{attribute 'qualified_only'}
{attribute 'TcHmiSymbol' := 'true'}
VAR_GLOBAL
	
	bStartWrite : BOOL;
	bGeneratePDF: BOOL;
	bGeneratePDF2: BOOL;
	bStartRead: BOOL;
	bPreview: BOOL;
	localPDF : STRING;
	testPath : T_MaxString;
	sJsonOutput: STRING(100000);
	stReportHead: ST_ReportInfo;
	
(***** SQL Commands ***********************************************************************************)

//RUN CMDS	
isrtRun: STRING(5000) := 'INSERT INTO [dbo].[RUNS] ( [analyst], [comment], [softwareVersion], [sysMasterRevision], [sysSettingsRevision], [meterVelocity], [runVelocity], [emptyTubesFactor], [fillTubesFactor], [solvent1NameRevision], [solvent2NameRevision], [solvent3NameRevision], [solvent4NameRevision], [timeEventStarted], [timeEventCompleted], [methodID], [CalibrationNo]) VALUES ( $'#1#$', $'#2#$', $'#3#$', $'#4#$', $'#5#$', $'#6#$', $'#7#$', $'#8#$', $'#9#$', $'#10#$', $'#11#$', $'#12#$', $'#13#$', $'#14#$', $'#15#$', #16#, #17#) ';
slctLastRun: STRING(1000) := 'SELECT TOP 1 [runNo], [analyst], [comment], [softwareVersion], [sysMasterRevision], [sysSettingsRevision], [meterVelocity], [runVelocity], [emptyTubesFactor], [fillTubesFactor], [solvent1NameRevision], [solvent2NameRevision], [solvent3NameRevision], [solvent4NameRevision], [timeEventStarted], [timeEventCompleted], [methodID], [CalibrationNo] FROM [dbo].[RUNS] ORDER BY [runNo] DESC;';

//METHOD CMDS
slctAllMethods: STRING(5000) := 'SELECT [methodName], [methodRevision] FROM [dbo].[METHODS] ';
slctAllActvMethod: STRING(5000) := 'SELECT [methodName], [methodRevision] FROM [dbo].[METHODS] WHERE [methodStatus] = $'activated$'';
slctMethod: STRING(5000) := 'SELECT [methodName], [methodRevision], [methodCreatedBy], [methodCreatedOn], [solvent_R1], [solvent_R2], [solvent_W1], [solvent_W2], [time_R1], [time_R2], [time_W1], [time_W2], [velocity_R1], [velocity_R2], [velocity_W1], [velocity_W2], [soakTime], [agitate_1_Time], [agitate_2_Time], [vialsToFill], [vialPrimeVol], [vial_1_FillVol], [vial_2_4_FillVol], [airDryTime], [methodID], [methodStatus] FROM [dbo].[METHODS] WHERE [methodName] = $'#1#$' AND [methodRevision] = $'#2#$' ';
slctVD: STRING(5000) := 'SELECT [VD_ID], [pump], [stage], [rinse1], [rinse2], [wash1], [wash2], [methodID] FROM [dbo].[VOLUME_DATA] WHERE [methodID] = #1# ';
slctMethodID: STRING(5000) := 'SELECT TOP 1 [methodID] FROM [dbo].[METHODS] WHERE [methodName] = $'#1#$' ORDER BY [methodID] DESC;';
isrtNewMethod: STRING(5000) := 'INSERT INTO [dbo].[METHODS] ( [methodName], [methodRevision], [methodCreatedBy], [methodCreatedOn], [solvent_R1], [solvent_R2], [solvent_W1], [solvent_W2], [time_R1], [time_R2], [time_W1], [time_W2], [velocity_R1], [velocity_R2], [velocity_W1], [velocity_W2], [soakTime], [agitate_1_Time], [agitate_2_Time], [vialsToFill], [vialPrimeVol], [vial_1_FillVol], [vial_2_4_FillVol], [airDryTime], [methodStatus]) VALUES ( $'#1#$', $'#2#$', $'#3#$', $'#4#$', $'#5#$', $'#6#$', $'#7#$', $'#8#$', $'#9#$', $'#10#$', $'#11#$', $'#12#$', $'#13#$', $'#14#$', $'#15#$', $'#16#$', $'#17#$', $'#18#$', $'#19#$', $'#20#$', $'#21#$', $'#22#$', $'#23#$', $'#24#$', $'#25#$') ';
isrtVD: string(5000) := 'INSERT INTO [dbo].[VOLUME_DATA] ( [pump], [stage], [rinse1], [rinse2], [wash1], [wash2], [methodID]) VALUES ( $'#1#$', $'#2#$', $'#3#$', $'#4#$', $'#5#$', $'#6#$', #7#) ';
updtDactvMethod: STRING(5000) := 'UPDATE [dbo].[METHODS] SET [methodStatus] = $'deactivated$' WHERE [methodName] = $'#1#$' AND [methodRevision] = $'#2#$'';

//CALIBRATION CMD
slctLastCalibID: T_Maxstring := 'SELECT TOP 1 [calibrationNo] FROM [dbo].[CALIBRATION_HEAD] ORDER BY [calibrationNo] DESC;';
slctLastCalib: STRING(5000) := 'SELECT TOP 1 [dateTime], [pumpNo], [step], [tareWt], [grossWt], [netVolume], [netWt], [targetVolume], [differencePercent], [criteria], [pumpRevs], [CalibrationNo] FROM [dbo].[CALIBRATION] ORDER BY [calibrationNo] DESC; ';
isrtCalib: STRING(5000) := 'INSERT INTO [dbo].[CALIBRATION_HEAD] ( [userID], [density], [solventNo], [solventRevision], [allowableFail], [replicates], [callInterval], [sysRevisionNo]) VALUES ( $'#1#$', $'#2#$', $'#3#$', $'#4#$', $'#5#$', $'#6#$', $'#7#$', #8#) ';
isrtCalibValues: STRING(5000) := 'INSERT INTO [dbo].[CALIBRATION] ( [dateTime], [pumpNo], [step], [tareWt], [grossWt], [netVolume], [netWt], [targetVolume], [differencePercent], [criteria], [pumpRevs], [CalibrationNo]) VALUES ( $'#1#$', $'#2#$', $'#3#$', $'#4#$', $'#5#$', $'#6#$', $'#7#$', $'#8#$', $'#9#$', $'#10#$', $'#11#$', #12#) ';
dltCalibHead : STRING(500) :='DELETE FROM [dbo].[CALIBRATION_HEAD] WHERE [calibrationNo] = #1#';

//SYSTEM CMD
slctLastSys: STRING(5000) := 'SELECT TOP 1 [gen_SealAndPump], [cal_AcceptanceCriteria], [cal_AllowableFail], [cal_Replicates], [cal_PumpCallIntervalDays], [cal_CloseAppOnCompletation], [AirDryTimeOnCompletation], [lkt_AllowableLeakTestFail], [lkt_LeakTestBuildupTime], [lkt_LeakTestHoldTime], [lkt_LeakTestPressure], [mec_PlatesClosedPosition], [mec_PlatesDryPosition], [mec_PlatesVelocity], [mec_MaxCurrentFastDown], [mec_MaxCurrentSlowDown], [mec_MaxCurrentSlowUp], [pmp_MeterVelocity], [pmp_RunVelocity], [pmp_EmptyFactor], [pmp_FillSolventTubesFactor], [smp_AboveCalibration], [smp_VialSetSpacing], [smp_IntoResBottom], [smp_IntoResDispense], [smp_IntoResWeigh], [smp_IntoVials], [sec_DisplayManualControl], [sec_CheckLogonEachRun], [createdBy], [createdDate], [sysRevisionNo], [smp_AboveVialSet1], [smp_IntoWaste] FROM [dbo].[SYSTEM] ORDER BY [sysRevisionNo] DESC; ';
slctAllSys: STRING(5000) := 'SELECT [gen_SealAndPump], [cal_AcceptanceCriteria], [cal_AllowableFail], [cal_Replicates], [cal_PumpCallIntervalDays], [cal_CloseAppOnCompletation], [AirDryTimeOnCompletation], [lkt_AllowableLeakTestFail], [lkt_LeakTestBuildupTime], [lkt_LeakTestHoldTime], [lkt_LeakTestPressure], [mec_PlatesClosedPosition], [mec_PlatesDryPosition], [mec_PlatesVelocity], [mec_MaxCurrentFastDown], [mec_MaxCurrentSlowDown], [mec_MaxCurrentSlowUp], [pmp_MeterVelocity], [pmp_RunVelocity], [pmp_EmptyFactor], [pmp_FillSolventTubesFactor], [smp_AboveCalibration], [smp_VialSetSpacing], [smp_IntoResBottom], [smp_IntoResDispense], [smp_IntoResWeigh], [smp_IntoVials], [sec_DisplayManualControl], [sec_CheckLogonEachRun], [createdBy], [createdDate], [sysRevisionNo], [smp_AboveVialSet1], [smp_IntoWaste] FROM [dbo].[SYSTEM] ORDER BY [sysRevisionNo] DESC; ';
isrtSys: STRING(5000) := 'INSERT INTO [dbo].[SYSTEM] ( [gen_SealAndPump], [cal_AcceptanceCriteria], [cal_AllowableFail], [cal_Replicates], [cal_PumpCallIntervalDays], [cal_CloseAppOnCompletation], [AirDryTimeOnCompletation], [lkt_AllowableLeakTestFail], [lkt_LeakTestBuildupTime], [lkt_LeakTestHoldTime], [lkt_LeakTestPressure], [mec_PlatesClosedPosition], [mec_PlatesDryPosition], [mec_PlatesVelocity], [mec_MaxCurrentFastDown], [mec_MaxCurrentSlowDown], [mec_MaxCurrentSlowUp], [pmp_MeterVelocity], [pmp_RunVelocity], [pmp_EmptyFactor], [pmp_FillSolventTubesFactor], [smp_AboveCalibration], [smp_VialSetSpacing], [smp_IntoResBottom], [smp_IntoResDispense], [smp_IntoResWeigh], [smp_IntoVials], [sec_DisplayManualControl], [sec_CheckLogonEachRun], [createdBy], [createdDate], [smp_AboveVialSet1], [smp_IntoWaste]) VALUES ( $'#1#$', $'#2#$', $'#3#$', $'#4#$', $'#5#$', $'#6#$', $'#7#$', $'#8#$', $'#9#$', $'#10#$', $'#11#$', $'#12#$', $'#13#$', $'#14#$', $'#15#$', $'#16#$', $'#17#$', $'#18#$', $'#19#$', $'#20#$', $'#21#$', $'#22#$', $'#23#$', $'#24#$', $'#25#$', $'#26#$', $'#27#$', $'#28#$', $'#29#$', $'#30#$', $'#31#$', $'#32#$', $'#33#$') ';

//USERS CMD
isrtUser: STRING(5000) := 'INSERT INTO [dbo].[USERS] ( [userID], [acessLevel], [transactionType], [transactionDate], [transactedBy], [addDate], [enteredBy]) VALUES ( $'#1#$', $'#2#$', $'#3#$', $'#4#$', $'#5#$', $'#6#$', $'#7#$') ';
slctCurrentUser: STRING(5000) := 'SELECT [ID_user], [userID], [acessLevel], [transactionType], [transactionDate], [transactedBy], [addDate], [enteredBy] FROM (SELECT *, ROW_NUMBER() OVER (PARTITION BY [userID] ORDER BY TRY_CONVERT(datetime, [transactionDate], 113) DESC, [ID_user] DESC) AS rn FROM [dbo].[USERS] WHERE [transactionType] = $'Added$') t WHERE rn = 1 AND NOT EXISTS (SELECT 1 FROM [dbo].[USERS] r WHERE r.[userID] = t.[userID] AND r.[transactionType] = $'Removed$' AND TRY_CONVERT(datetime, r.[transactionDate], 113) > TRY_CONVERT(datetime, t.[transactionDate], 113));';
slctAllUsers: STRING(5000) := 'SELECT [ID_user], [userID], [acessLevel], [transactionType], [transactionDate], [transactedBy], [addDate], [enteredBy] FROM [dbo].[USERS] ';

//SOLVENTS
isrtSolvent: STRING(1000) := 'INSERT INTO [dbo].[SOLVENTS] ( [solventName1], [solventName2], [solventName3], [solventName4], [density1], [density2], [density3], [density4], [addedBy], [addedDate]) VALUES ( $'#1#$', $'#2#$', $'#3#$', $'#4#$', $'#5#$', $'#6#$', $'#7#$', $'#8#$', $'#9#$', $'#10#$') ';
slctSolvent: STRING(1000) := 'SELECT TOP 1 [SOLVENT_ID], [solventName1], [solventName2], [solventName3], [solventName4], [density1], [density2], [density3], [density4], [addedBy], [addedDate] FROM [dbo].[SOLVENTS] ORDER BY [SOLVENT_ID] DESC; ';
slctAllSolvents: STRING(1000) := 'SELECT [SOLVENT_ID], [solventName1], [solventName2], [solventName3], [solventName4], [density1], [density2], [density3], [density4], [addedBy], [addedDate] FROM [dbo].[SOLVENTS] ';

//LINEAR MOTORS
isrtLinear: STRING(1500) := 'INSERT INTO [dbo].[LINEAR] ( [pump1], [pump2], [pump3], [pump4], [pump5], [pump6], [pump7], [pump8], [pump9], [pump10], [changedBy], [changedOn]) VALUES ( $'#1#$', $'#2#$', $'#3#$', $'#4#$', $'#5#$', $'#6#$', $'#7#$', $'#8#$', $'#9#$', $'#10#$', $'#11#$', $'#12#$') ';
slctLinear: STRING(1000) := 'SELECT TOP 1 [ID_Linear], [pump1], [pump2], [pump3], [pump4], [pump5], [pump6], [pump7], [pump8], [pump9], [pump10] FROM [dbo].[LINEAR] ORDER BY [ID_Linear] DESC; ';

//PUMP CALIBRATION REPORT / HISTORY CMD
slctCalibReportList: STRING(5000) := 'SELECT TOP 50 [CalibrationNo], [userID], [solventNo], [sysRevisionNo] FROM [dbo].[PumpCalibrationHeader] ORDER BY [CalibrationNo] DESC;';
slctPumpCalibHeaderByNo: STRING(5000) := 'SELECT TOP 1 [CalibrationNo], [userID], [density], [solventNo], [solventRevision], [allowableFail], [replicates], [callInterval], [sysRevisionNo] FROM [dbo].[PumpCalibrationHeader] WHERE [CalibrationNo] = #1#;';
slctPumpCalibValuesByNo: STRING(5000) := 'SELECT [CalibrationNo], [dateTime], [pumpNo], [step], [tareWt], [grossWt], [netVolume], [netWt], [targetVolume], [differencePercent], [criteria], [pumpRevs] FROM [dbo].[PumpCalibrationValues] WHERE [CalibrationNo] = #1# ORDER BY [ID] ASC;';

slctCalibReportListFromValues: STRING(5000) := 'SELECT TOP 100 CAST(ISNULL([ReportType], $'$') AS VARCHAR(50)) AS [ReportType], CAST(ISNULL([ReportID], $'$') AS VARCHAR(50)) AS [ReportID], CAST(ISNULL([CreatedOn], $'$') AS VARCHAR(30)) AS [CreatedOn], CAST(ISNULL([CreatedBy], $'$') AS VARCHAR(50)) AS [CreatedBy], CAST(ISNULL([Description], $'$') AS VARCHAR(200)) AS [Description], CAST(ISNULL([sPrimaryKey], $'$') AS VARCHAR(50)) AS [sPrimaryKey] FROM [dbo].[vw_ReportList_PumpCalibration] ORDER BY CAST([ReportID] AS INT) DESC;';
slctMethodReportList: STRING(5000) := 'SELECT TOP 50 $'Method$' AS [ReportType], CAST([methodID] AS VARCHAR(50)) AS [ReportID], [methodCreatedOn] AS [CreatedOn], [methodCreatedBy] AS [CreatedBy], [methodName] + $' Rev $' + [methodRevision] AS [Description], CAST([methodID] AS VARCHAR(50)) AS [sPrimaryKey] FROM [dbo].[METHODS] ORDER BY [methodID] DESC;';
slctRunReportList: STRING(5000) := 'SELECT TOP 100 CAST(ISNULL($'Run$', $'$') AS VARCHAR(50)) AS [ReportType], CAST(ISNULL(CAST([runNo] AS VARCHAR(50)), $'$') AS VARCHAR(50)) AS [ReportID], CAST(ISNULL([timeEventCompleted], $'$') AS VARCHAR(30)) AS [CreatedOn], CAST(ISNULL([analyst], $'$') AS VARCHAR(50)) AS [CreatedBy], CAST(ISNULL($'Method ID $' + CAST([methodID] AS VARCHAR(20)) + $' / Cal $' + CAST([CalibrationNo] AS VARCHAR(20)) + CASE WHEN ISNULL([comment], $'$') = $'$' THEN $'$' ELSE $' - $' + [comment] END, $'$') AS VARCHAR(200)) AS [Description], CAST(ISNULL(CAST([runNo] AS VARCHAR(50)), $'$') AS VARCHAR(50)) AS [sPrimaryKey] FROM [dbo].[RUNS] ORDER BY [runNo] DESC;';
slctLinearReportList: STRING(5000) := 'SELECT TOP 50 $'Linear$' AS [ReportType], CAST([ID_Linear] AS VARCHAR(50)) AS [ReportID], $'$' AS [CreatedOn], $'$' AS [CreatedBy], $'Linear pump positions set $' + CAST([ID_Linear] AS VARCHAR(20)) AS [Description], CAST([ID_Linear] AS VARCHAR(50)) AS [sPrimaryKey] FROM [dbo].[LINEAR] ORDER BY [ID_Linear] DESC;';

// REPORT SCREEN LISTING AND SELECTING
slctPumpCalibHeaderByNo1: STRING(5000) := 'SELECT TOP 1 CAST($'Pump Calibration$' AS VARCHAR(50)) AS [sReportId], CAST(ISNULL([CalibrationNo], $'$') AS VARCHAR(30)) AS [sCalibrationNo], CAST(ISNULL([userID], $'$') AS VARCHAR(50)) AS [sUserId], CAST(ISNULL([density], $'$') AS VARCHAR(30)) AS [sDensity], CAST(ISNULL([solventNo], $'$') AS VARCHAR(30)) AS [sSolventNo], CAST(ISNULL([solventRevision], $'$') AS VARCHAR(30)) AS [sSolventRevision], CAST(ISNULL([sysRevisionNo], $'$') AS VARCHAR(30)) AS [sSysRevisionNo], CAST(ISNULL([allowableFail], $'$') AS VARCHAR(30)) AS [sAllowableFail], CAST(ISNULL([replicates], $'$') AS VARCHAR(30)) AS [sReplicates], CAST(ISNULL([callInterval], $'$') AS VARCHAR(30)) AS [sCallInterval], CAST($'$' AS VARCHAR(30)) AS [sCreatedAt] FROM [dbo].[CALIBRATION_HEAD] WHERE [CalibrationNo] = #1#;';
slctPumpCalibValuesByNo1: STRING(5000) := 'SELECT CAST(ISNULL([dateTime], $'$') AS VARCHAR(40)) AS [sDateTime], CAST(ISNULL([pumpNo], $'$') AS VARCHAR(10)) AS [sPumpNo], CAST(ISNULL([step], $'$') AS VARCHAR(20)) AS [sStep], CAST(ISNULL([tareWt], $'$') AS VARCHAR(30)) AS [sTareWt], CAST(ISNULL([grossWt], $'$') AS VARCHAR(30)) AS [sGrossWt], CAST(ISNULL([netWt], $'$') AS VARCHAR(30)) AS [sNetWt], CAST(ISNULL([netVolume], $'$') AS VARCHAR(30)) AS [sNetVolume], CAST(ISNULL([targetVolume], $'$') AS VARCHAR(30)) AS [sTargetVolume], CAST(ISNULL([differencePercent], $'$') AS VARCHAR(30)) AS [sDifferencePercent], CAST(ISNULL([criteria], $'$') AS VARCHAR(20)) AS [sCriteria], CAST(ISNULL([pumpRevs], $'$') AS VARCHAR(30)) AS [sPumpRevs] FROM [dbo].[CALIBRATION] WHERE [CalibrationNo] = #1# ORDER BY [Data_ID] ASC;';
slctSystemSettingsReportList: STRING(5000) := 'SELECT TOP 100 CAST([ReportType] AS VARCHAR(50)) AS [ReportType], CAST([ReportID] AS VARCHAR(50)) AS [ReportID], CAST([CreatedOn] AS VARCHAR(30)) AS [CreatedOn], CAST([CreatedBy] AS VARCHAR(50)) AS [CreatedBy], CAST([Description] AS VARCHAR(200)) AS [Description], CAST([sPrimaryKey] AS VARCHAR(50)) AS [sPrimaryKey] FROM [dbo].[vw_ReportList_SystemSettings] ORDER BY CAST([ReportID] AS INT) DESC;';
slctSystemSettingsByRevision: STRING(5000) := 'SELECT TOP 1 CAST([gen_SealAndPump] AS VARCHAR(100)) AS [sGenSealAndPump], CAST([cal_AcceptanceCriteria] AS VARCHAR(100)) AS [sCalAcceptanceCriteria], CAST([cal_AllowableFail] AS VARCHAR(100)) AS [sCalAllowableFail], CAST([cal_Replicates] AS VARCHAR(100)) AS [sCalReplicates], CAST([cal_PumpCallIntervalDays] AS VARCHAR(100)) AS [sCalPumpCallIntervalDays], CAST([cal_CloseAppOnCompletation] AS VARCHAR(100)) AS [sCalCloseAppOnCompletion], CAST([AirDryTimeOnCompletation] AS VARCHAR(100)) AS [sAirDryTimeOnCompletion], CAST([lkt_AllowableLeakTestFail] AS VARCHAR(100)) AS [sLktAllowableLeakTestFail], CAST([lkt_LeakTestBuildupTime] AS VARCHAR(100)) AS [sLktLeakTestBuildUpTime], CAST([lkt_LeakTestHoldTime] AS VARCHAR(100)) AS [sLktLeakTestHoldTime], CAST([lkt_LeakTestPressure] AS VARCHAR(100)) AS [sLktLeakTestPressure], CAST([mec_PlatesClosedPosition] AS VARCHAR(100)) AS [sMecPlatesClosedPosition], CAST([mec_PlatesDryPosition] AS VARCHAR(100)) AS [sMecPlatesDryPosition], CAST([mec_PlatesVelocity] AS VARCHAR(100)) AS [sMecPlatesVelocity], CAST([mec_MaxCurrentFastDown] AS VARCHAR(100)) AS [sMecMaxCurrentFastDown], CAST([mec_MaxCurrentSlowDown] AS VARCHAR(100)) AS [sMecMaxCurrentSlowDown], CAST([mec_MaxCurrentSlowUp] AS VARCHAR(100)) AS [sMecMaxCurrentSlowUp], CAST([pmp_MeterVelocity] AS VARCHAR(100)) AS [sPmpMeterVelocity], CAST([pmp_RunVelocity] AS VARCHAR(100)) AS [sPmpRunVelocity], CAST([pmp_EmptyFactor] AS VARCHAR(100)) AS [sPmpEmptyFactor], CAST([pmp_FillSolventTubesFactor] AS VARCHAR(100)) AS [sPmpFillSolventTubesFactor], CAST([smp_AboveCalibration] AS VARCHAR(100)) AS [sSmpAboveCalibration], CAST([smp_VialSetSpacing] AS VARCHAR(100)) AS [sSmpVialSetSpacing], CAST([smp_IntoResBottom] AS VARCHAR(100)) AS [sSmpIntoResBottom], CAST([smp_IntoResDispense] AS VARCHAR(100)) AS [sSmpIntoResDispense], CAST([smp_IntoResWeigh] AS VARCHAR(100)) AS [sSmpIntoResWeigh], CAST([smp_IntoVials] AS VARCHAR(100)) AS [sSmpIntoVials], CAST([smp_IntoWaste] AS VARCHAR(100)) AS [sSmpIntoWaste], CAST([sec_DisplayManualControl] AS VARCHAR(100)) AS [sSecDisplayManualControl], CAST([sec_CheckLogonEachRun] AS VARCHAR(100)) AS [sSecCheckLogonEachRun], CAST([createdBy] AS VARCHAR(100)) AS [sCreatedBy], CAST([createdDate] AS VARCHAR(100)) AS [sCreatedDate], CAST([sysRevisionNo] AS VARCHAR(30)) AS [sSysRevisionNo] FROM [dbo].[SYSTEM] WHERE [sysRevisionNo] = #1#;';
slctMethodReportSearchLatest : STRING(5000) := 'SELECT TOP 100 CAST(ISNULL([ReportType], $'$') AS VARCHAR(50)) AS [ReportType], CAST(ISNULL([ReportID], $'$') AS VARCHAR(50)) AS [ReportID], CAST(ISNULL([CreatedOn], $'$') AS VARCHAR(30)) AS [CreatedOn], CAST(ISNULL([CreatedBy], $'$') AS VARCHAR(50)) AS [CreatedBy], CAST(ISNULL([Description], $'$') AS VARCHAR(200)) AS [Description], CAST(ISNULL([sPrimaryKey], $'$') AS VARCHAR(50)) AS [sPrimaryKey] FROM [dbo].[vw_ReportList_Recipe] ORDER BY CAST([ReportID] AS INT) DESC;';
slctMethodHeaderByID : STRING(5000) := 'SELECT TOP 1 CAST(ISNULL([methodName], $'$') AS VARCHAR(100)) AS [methodName], CAST(ISNULL([methodRevision], $'$') AS VARCHAR(100)) AS [methodRevision], CAST(ISNULL([methodCreatedBy], $'$') AS VARCHAR(100)) AS [methodCreatedBy], CAST(ISNULL([methodCreatedOn], $'$') AS VARCHAR(100)) AS [methodCreatedOn], CAST(ISNULL([solvent_R1], $'$') AS VARCHAR(100)) AS [solvent_R1], CAST(ISNULL([solvent_R2], $'$') AS VARCHAR(100)) AS [solvent_R2], CAST(ISNULL([solvent_W1], $'$') AS VARCHAR(100)) AS [solvent_W1], CAST(ISNULL([solvent_W2], $'$') AS VARCHAR(100)) AS [solvent_W2], CAST(ISNULL([time_R1], $'$') AS VARCHAR(100)) AS [time_R1], CAST(ISNULL([time_R2], $'$') AS VARCHAR(100)) AS [time_R2], CAST(ISNULL([time_W1], $'$') AS VARCHAR(100)) AS [time_W1], CAST(ISNULL([time_W2], $'$') AS VARCHAR(100)) AS [time_W2], CAST(ISNULL([velocity_R1], $'$') AS VARCHAR(100)) AS [velocity_R1], CAST(ISNULL([velocity_R2], $'$') AS VARCHAR(100)) AS [velocity_R2], CAST(ISNULL([velocity_W1], $'$') AS VARCHAR(100)) AS [velocity_W1], CAST(ISNULL([velocity_W2], $'$') AS VARCHAR(100)) AS [velocity_W2], CAST(ISNULL([soakTime], $'$') AS VARCHAR(100)) AS [soakTime], CAST(ISNULL([agitate_1_Time], $'$') AS VARCHAR(100)) AS [agitate_1_Time], CAST(ISNULL([agitate_2_Time], $'$') AS VARCHAR(100)) AS [agitate_2_Time], CAST(ISNULL([vialsToFill], $'$') AS VARCHAR(100)) AS [vialsToFill], CAST(ISNULL([vialPrimeVol], $'$') AS VARCHAR(100)) AS [vialPrimeVol], CAST(ISNULL([vial_1_FillVol], $'$') AS VARCHAR(100)) AS [vial_1_FillVol], CAST(ISNULL([vial_2_4_FillVol], $'$') AS VARCHAR(100)) AS [vial_2_4_FillVol], CAST(ISNULL([airDryTime], $'$') AS VARCHAR(100)) AS [airDryTime], ISNULL([methodID], 0) AS [methodID], CAST(ISNULL([methodStatus], $'$') AS VARCHAR(100)) AS [methodStatus] FROM [dbo].[METHODS] WHERE [methodID] = #1#;';
slctMethodVolumeByID : STRING(5000) := 'SELECT ISNULL([VD_ID], 0) AS [VD_ID], CAST(ISNULL([pump], $'$') AS VARCHAR(100)) AS [pump], CAST(ISNULL([stage], $'$') AS VARCHAR(100)) AS [stage], CAST(ISNULL([rinse1], $'$') AS VARCHAR(100)) AS [rinse1], CAST(ISNULL([rinse2], $'$') AS VARCHAR(100)) AS [rinse2], CAST(ISNULL([wash1], $'$') AS VARCHAR(100)) AS [wash1], CAST(ISNULL([wash2], $'$') AS VARCHAR(100)) AS [wash2], ISNULL([methodID], 0) AS [methodID] FROM [dbo].[VOLUME_DATA] WHERE [methodID] = #1# ORDER BY [VD_ID] ASC;';
slctPostRunHeaderByID : STRING(5000) := 'SELECT TOP 1 ISNULL([runNo], 0) AS [runNo], CAST(ISNULL([analyst], $'$') AS VARCHAR(100)) AS [analyst], CAST(ISNULL([comment], $'$') AS VARCHAR(100)) AS [comment], CAST(ISNULL([softwareVersion], $'$') AS VARCHAR(100)) AS [softwareVersion], CAST(ISNULL([sysMasterRevision], $'$') AS VARCHAR(100)) AS [sysMasterRevision], CAST(ISNULL([sysSettingsRevision], $'$') AS VARCHAR(100)) AS [sysSettingsRevision], CAST(ISNULL([meterVelocity], $'$') AS VARCHAR(100)) AS [meterVelocity], CAST(ISNULL([runVelocity], $'$') AS VARCHAR(100)) AS [runVelocity], CAST(ISNULL([emptyTubesFactor], $'$') AS VARCHAR(100)) AS [emptyTubesFactor], CAST(ISNULL([fillTubesFactor], $'$') AS VARCHAR(100)) AS [fillTubesFactor], CAST(ISNULL([solvent1NameRevision], $'$') AS VARCHAR(100)) AS [solvent1NameRevision], CAST(ISNULL([solvent2NameRevision], $'$') AS VARCHAR(100)) AS [solvent2NameRevision], CAST(ISNULL([solvent3NameRevision], $'$') AS VARCHAR(100)) AS [solvent3NameRevision], CAST(ISNULL([solvent4NameRevision], $'$') AS VARCHAR(100)) AS [solvent4NameRevision], CAST(ISNULL([timeEventStarted], $'$') AS VARCHAR(100)) AS [timeEventStarted], CAST(ISNULL([timeEventCompleted], $'$') AS VARCHAR(100)) AS [timeEventCompleted], ISNULL([methodID], 0) AS [methodID], ISNULL([CalibrationNo], 0) AS [CalibrationNo] FROM [dbo].[RUNS] WHERE [runNo] = #1#;';
slctPostRunMethodHeaderByID : STRING(5000) := 'SELECT TOP 1 CAST(ISNULL([methodName], $'$') AS VARCHAR(100)) AS [methodName], CAST(ISNULL([methodRevision], $'$') AS VARCHAR(100)) AS [methodRevision], CAST(ISNULL([methodCreatedBy], $'$') AS VARCHAR(100)) AS [methodCreatedBy], CAST(ISNULL([methodCreatedOn], $'$') AS VARCHAR(100)) AS [methodCreatedOn], CAST(ISNULL([solvent_R1], $'$') AS VARCHAR(100)) AS [solvent_R1], CAST(ISNULL([solvent_R2], $'$') AS VARCHAR(100)) AS [solvent_R2], CAST(ISNULL([solvent_W1], $'$') AS VARCHAR(100)) AS [solvent_W1], CAST(ISNULL([solvent_W2], $'$') AS VARCHAR(100)) AS [solvent_W2], CAST(ISNULL([time_R1], $'$') AS VARCHAR(100)) AS [time_R1], CAST(ISNULL([time_R2], $'$') AS VARCHAR(100)) AS [time_R2], CAST(ISNULL([time_W1], $'$') AS VARCHAR(100)) AS [time_W1], CAST(ISNULL([time_W2], $'$') AS VARCHAR(100)) AS [time_W2], CAST(ISNULL([velocity_R1], $'$') AS VARCHAR(100)) AS [velocity_R1], CAST(ISNULL([velocity_R2], $'$') AS VARCHAR(100)) AS [velocity_R2], CAST(ISNULL([velocity_W1], $'$') AS VARCHAR(100)) AS [velocity_W1], CAST(ISNULL([velocity_W2], $'$') AS VARCHAR(100)) AS [velocity_W2], CAST(ISNULL([soakTime], $'$') AS VARCHAR(100)) AS [soakTime], CAST(ISNULL([agitate_1_Time], $'$') AS VARCHAR(100)) AS [agitate_1_Time], CAST(ISNULL([agitate_2_Time], $'$') AS VARCHAR(100)) AS [agitate_2_Time], CAST(ISNULL([vialsToFill], $'$') AS VARCHAR(100)) AS [vialsToFill], CAST(ISNULL([vialPrimeVol], $'$') AS VARCHAR(100)) AS [vialPrimeVol], CAST(ISNULL([vial_1_FillVol], $'$') AS VARCHAR(100)) AS [vial_1_FillVol], CAST(ISNULL([vial_2_4_FillVol], $'$') AS VARCHAR(100)) AS [vial_2_4_FillVol], CAST(ISNULL([airDryTime], $'$') AS VARCHAR(100)) AS [airDryTime], ISNULL([methodID], 0) AS [methodID], CAST(ISNULL([methodStatus], $'$') AS VARCHAR(100)) AS [methodStatus] FROM [dbo].[METHODS] WHERE [methodID] = #1#;';
slctPostRunVolumeByMethodID : STRING(5000) := 'SELECT ISNULL([VD_ID], 0) AS [VD_ID], CAST(ISNULL([pump], $'$') AS VARCHAR(100)) AS [pump], CAST(ISNULL([stage], $'$') AS VARCHAR(100)) AS [stage], CAST(ISNULL([rinse1], $'$') AS VARCHAR(100)) AS [rinse1], CAST(ISNULL([rinse2], $'$') AS VARCHAR(100)) AS [rinse2], CAST(ISNULL([wash1], $'$') AS VARCHAR(100)) AS [wash1], CAST(ISNULL([wash2], $'$') AS VARCHAR(100)) AS [wash2], ISNULL([methodID], 0) AS [methodID] FROM [dbo].[VOLUME_DATA] WHERE [methodID] = #1# ORDER BY [VD_ID] ASC;';
slctLinearReportSearch : STRING(5000) := 'SELECT TOP 100 CAST(ISNULL([ReportType], $'$') AS VARCHAR(50)) AS [ReportType], CAST(ISNULL([ReportID], $'$') AS VARCHAR(50)) AS [ReportID], CAST(ISNULL([CreatedOn], $'$') AS VARCHAR(30)) AS [CreatedOn], CAST(ISNULL([CreatedBy], $'$') AS VARCHAR(50)) AS [CreatedBy], CAST(ISNULL([Description], $'$') AS VARCHAR(200)) AS [Description], CAST(ISNULL([sPrimaryKey], $'$') AS VARCHAR(50)) AS [sPrimaryKey] FROM [dbo].[vw_ReportList_Linear] ORDER BY CAST([ReportID] AS INT) DESC;';
slctLinearByID : STRING(5000) := 'SELECT TOP 1 ISNULL([ID_Linear], 0) AS [ID_Linear], CAST(ISNULL([pump1], $'$') AS VARCHAR(100)) AS [pump1], CAST(ISNULL([pump2], $'$') AS VARCHAR(100)) AS [pump2], CAST(ISNULL([pump3], $'$') AS VARCHAR(100)) AS [pump3], CAST(ISNULL([pump4], $'$') AS VARCHAR(100)) AS [pump4], CAST(ISNULL([pump5], $'$') AS VARCHAR(100)) AS [pump5], CAST(ISNULL([pump6], $'$') AS VARCHAR(100)) AS [pump6], CAST(ISNULL([pump7], $'$') AS VARCHAR(100)) AS [pump7], CAST(ISNULL([pump8], $'$') AS VARCHAR(100)) AS [pump8], CAST(ISNULL([pump9], $'$') AS VARCHAR(100)) AS [pump9], CAST(ISNULL([pump10], $'$') AS VARCHAR(100)) AS [pump10], CAST(ISNULL([changedBy], $'$') AS VARCHAR(100)) AS [changedBy], CAST(ISNULL([changedOn], $'$') AS VARCHAR(100)) AS [changedOn] FROM [dbo].[LINEAR] WHERE [ID_Linear] = #1#;';

// REPORT SCREEN FILTERING
slctCalibReportListByDate : STRING(5000) := 'SELECT TOP 100 CAST(ISNULL([ReportType], $'$') AS VARCHAR(50)) AS [ReportType], CAST(ISNULL([ReportID], $'$') AS VARCHAR(50)) AS [ReportID], CAST(ISNULL([CreatedOn], $'$') AS VARCHAR(30)) AS [CreatedOn], CAST(ISNULL([CreatedBy], $'$') AS VARCHAR(50)) AS [CreatedBy], CAST(ISNULL([Description], $'$') AS VARCHAR(200)) AS [Description], CAST(ISNULL([sPrimaryKey], $'$') AS VARCHAR(50)) AS [sPrimaryKey] FROM [dbo].[vw_ReportList_PumpCalibration] WHERE TRY_PARSE([CreatedOn] AS datetime USING $'en-GB$') >= #1# AND TRY_PARSE([CreatedOn] AS datetime USING $'en-GB$') <= #2# ORDER BY TRY_PARSE([CreatedOn] AS datetime USING $'en-GB$') DESC, CAST([ReportID] AS INT) DESC;';
slctSystemSettingsReportListByDate : STRING(5000) := 'SELECT TOP 100 CAST(ISNULL([ReportType], $'$') AS VARCHAR(50)) AS [ReportType], CAST(ISNULL([ReportID], $'$') AS VARCHAR(50)) AS [ReportID], CAST(ISNULL([CreatedOn], $'$') AS VARCHAR(30)) AS [CreatedOn], CAST(ISNULL([CreatedBy], $'$') AS VARCHAR(50)) AS [CreatedBy], CAST(ISNULL([Description], $'$') AS VARCHAR(200)) AS [Description], CAST(ISNULL([sPrimaryKey], $'$') AS VARCHAR(50)) AS [sPrimaryKey] FROM [dbo].[vw_ReportList_SystemSettings] WHERE TRY_PARSE([CreatedOn] AS datetime USING $'en-GB$') >= #1# AND TRY_PARSE([CreatedOn] AS datetime USING $'en-GB$') <= #2# ORDER BY TRY_PARSE([CreatedOn] AS datetime USING $'en-GB$') DESC, CAST([ReportID] AS INT) DESC;';
slctMethodReportSearchLatestByDate : STRING(5000) := 'SELECT TOP 100 CAST(ISNULL([ReportType], $'$') AS VARCHAR(50)) AS [ReportType], CAST(ISNULL([ReportID], $'$') AS VARCHAR(50)) AS [ReportID], CAST(ISNULL([CreatedOn], $'$') AS VARCHAR(30)) AS [CreatedOn], CAST(ISNULL([CreatedBy], $'$') AS VARCHAR(50)) AS [CreatedBy], CAST(ISNULL([Description], $'$') AS VARCHAR(200)) AS [Description], CAST(ISNULL([sPrimaryKey], $'$') AS VARCHAR(50)) AS [sPrimaryKey] FROM [dbo].[vw_ReportList_Recipe] WHERE TRY_PARSE(REPLACE([CreatedOn], $'D#$', $'$') AS datetime USING $'en-GB$') >= #1# AND TRY_PARSE(REPLACE([CreatedOn], $'D#$', $'$') AS datetime USING $'en-GB$') <= #2# ORDER BY TRY_PARSE(REPLACE([CreatedOn], $'D#$', $'$') AS datetime USING $'en-GB$') DESC, CAST([ReportID] AS INT) DESC;';
slctLinearReportListByDate : STRING(5000) := 'SELECT TOP 100 CAST(ISNULL([ReportType], $'$') AS VARCHAR(50)) AS [ReportType], CAST(ISNULL([ReportID], $'$') AS VARCHAR(50)) AS [ReportID], CAST(ISNULL([CreatedOn], $'$') AS VARCHAR(30)) AS [CreatedOn], CAST(ISNULL([CreatedBy], $'$') AS VARCHAR(50)) AS [CreatedBy], CAST(ISNULL([Description], $'$') AS VARCHAR(200)) AS [Description], CAST(ISNULL([sPrimaryKey], $'$') AS VARCHAR(50)) AS [sPrimaryKey] FROM [dbo].[vw_ReportList_Linear] WHERE TRY_PARSE([CreatedOn] AS datetime USING $'en-GB$') >= #1# AND TRY_PARSE([CreatedOn] AS datetime USING $'en-GB$') <= #2# ORDER BY TRY_PARSE([CreatedOn] AS datetime USING $'en-GB$') DESC, CAST([ReportID] AS INT) DESC;';

//CURRENT REPORTS
slctLastLinear : STRING(5000) := 'SELECT TOP 1 ISNULL([ID_Linear], 0) AS [ID_Linear], CAST(ISNULL([pump1], $'$') AS VARCHAR(100)) AS [pump1], CAST(ISNULL([pump2], $'$') AS VARCHAR(100)) AS [pump2], CAST(ISNULL([pump3], $'$') AS VARCHAR(100)) AS [pump3], CAST(ISNULL([pump4], $'$') AS VARCHAR(100)) AS [pump4], CAST(ISNULL([pump5], $'$') AS VARCHAR(100)) AS [pump5], CAST(ISNULL([pump6], $'$') AS VARCHAR(100)) AS [pump6], CAST(ISNULL([pump7], $'$') AS VARCHAR(100)) AS [pump7], CAST(ISNULL([pump8], $'$') AS VARCHAR(100)) AS [pump8], CAST(ISNULL([pump9], $'$') AS VARCHAR(100)) AS [pump9], CAST(ISNULL([pump10], $'$') AS VARCHAR(100)) AS [pump10], CAST(ISNULL([changedBy], $'$') AS VARCHAR(100)) AS [changedBy], CAST(ISNULL([changedOn], $'$') AS VARCHAR(100)) AS [changedOn] FROM [dbo].[LINEAR] ORDER BY [ID_Linear] DESC;';

(******************************************************************************************************)

(***** Pump Calibration Report Variables **************************************************************)

bBuildPCR			: BOOL;
stParameter_PCR		: ST_Parameters_PCR;
astData_PCR	  		: ARRAY[1..100] OF ST_Data_PCR;
lastCalibID			: ARRAY[0..1] OF INT;
lastCalibData		: array[1..100] of ST_Data_PCR;


(******************************************************************************************************)
	
(***** Post-Run Report Variables **********************************************************************)

bBuildPRRW		: BOOL;
stPostRunReport	: ARRAY[0..5] OF ST_PostRunReport;
lastRunID		: ARRAY[0..1] OF INT;
stPostRunInfo	: ST_PostRunReport;
runIsDone		: BOOL;

(******************************************************************************************************)

(***** User History Report Variables ******************************************************************)

bBuildUHR	   : BOOL;
astData_UHR	   : ARRAY[0..100] OF ST_Data_UHR;

(******************************************************************************************************)

(***** Current Users List Variables *****************************************************************)

bBuildCUL	   : BOOL;
astData_CUL	   : ARRAY[0..1000] OF ST_Data_CUL;

(******************************************************************************************************)

(***** Method Report Variables ************************************************************************)

bBuildMR			: BOOL;
stParameter_MR		: ST_Parameters_MR;
astVolData			: ARRAY[1..10] OF ST_VolumeData;
listOfMethod		: ARRAY[1..500] OF ST_ListMethod;
methodName			: STRING;
methodRevision		: STRING;
lastMethodID		: INT;
arrCompleteMethod	: ARRAY[1..100] OF ST_CompleteMethod;

(******************************************************************************************************)

(***** System Parameters Variables ********************************************************************)

stSysParameters	: ST_SysParameters;
listAllSystem	: ARRAY[0..500] OF ST_SysParameters;

(******************************************************************************************************)

(***** Solvents Variables *****************************************************************************)

stSolvents		: ST_Solvents;
listSolvents	: ARRAY[0..500] OF ST_Solvents;

(******************************************************************************************************)

(***** Linear Motors Variables *****************************************************************************)

stLinearMotors	: ST_LinearMotors;

(******************************************************************************************************)

(***** List Reports hmi *****************************************************************************)

aCalibReportList : ARRAY[1..100] OF ST_CalibrationReportListItem;

(******************************************************************************************************)

END_VAR

(* stored: Version 1.1.0.1, ProductVersion 3.1.4024.15
   GVL GVL_DB: Id {b6405db0-d623-4e3b-8d34-c8eb4e42140d} *)
